PROGRAM MAIN_1
VAR
	// trigger command execution for Postman-Echo samples
	
	
	fbMHS :  FB_MHS ;
	
	
	
	
END_VAR

fbMHS();

END_PROGRAM

(* stored: Version 1.1.0.1, ProductVersion 3.1.4024.3
   POU MAIN_1: Id {8a4442c4-294e-495c-aa76-75ff5f556fbf}, SpecialFunc None *)
